FUNCTION_BLOCK FB_MqttLight EXTENDS FB_Light IMPLEMENTS I_MqttMessageReceiver, I_MqttDeviceDiscoveryProvider
VAR_INPUT
END_VAR
VAR_OUTPUT
END_VAR
VAR
	rMqttController: REFERENCE TO FB_MqttController;
	fbDeviceDiscovery : FB_MqttLightDiscovery;
	sStateTopic: STRING(255); // The topic to publish the state to
	sCommandTopic : STRING(255);
	sCmdOnPayload: STRING(10); // The text which is published if On() is called
	sCmdOffPayload: STRING(10); // The test which is published if Off() is called
	sStateOnPayload: STRING(10); // The text which is published if On() is called
	sStateOffPayload: STRING(10); // The test which is published if Off() is called
END_VAR

METHOD FB_init : BOOL
VAR_INPUT
	bInitRetains : BOOL; // if TRUE, the retain variables are initialized (warm start / cold start)
	bInCopyCode : BOOL;  // if TRUE, the instance afterwards gets moved into the copy code (online change)
	rMqttController : REFERENCE TO FB_MqttController;
	sMainTopic : STRING(255); // The topic to publish
	sIdentifier : STRING(20);
	sName : STRING(30);
END_VAR
VAR
	stDevInfo : ST_MqttDeviceInformation;
	stDevConfig : ST_MqttLightConfiguration;
END_VAR
THIS^.rMqttController REF= rMqttController;

THIS^.sStateTopic := CONCAT(STR1 := sMainTopic, STR2 := '/');
THIS^.sStateTopic := CONCAT(STR1 := THIS^.sStateTopic, STR2 := GVL_MQTT_CONST.TOPIC_STATE);
THIS^.sCommandTopic := CONCAT(STR1 := sMainTopic, STR2 := '/');
THIS^.sCommandTopic := CONCAT(STR1 := THIS^.sCommandTopic, STR2 := GVL_MQTT_CONST.TOPIC_COMMAND);

THIS^.fbDeviceDiscovery.SetMqttClient(rMqttClient := THIS^.rMqttController.MqttClient);
THIS^.fbDeviceDiscovery.NodeId := GVL_MQTT_CONST.DEV_DISCOVER_NODEID;
THIS^.fbDeviceDiscovery.ObjectId := sIdentifier;

stDevConfig.command_topic := THIS^.sCommandTopic;
stDevConfig.state_topic := THIS^.sStateTopic;
stDevConfig.unique_id := sIdentifier;
stDevConfig.name := sName;
THIS^.fbDeviceDiscovery.Configuration := stDevConfig;

stDevInfo.identifiers := sIdentifier;
stDevInfo.manufacturer := GVL_MQTT_CONST.DEV_DISCOVER_MANUFACTURER;
stDevInfo.model := 'FB_MqttLight';
stDevInfo.sw_version := GVL_CONST.SW_VERSION;
stDevInfo.name := sName;
THIS^.fbDeviceDiscovery.DeviceInformation := stDevInfo;

THIS^.rMqttController.RegisterMqttMessageReceive(iMqttMessageReceiver := THIS^, sTopic := sCommandTopic);
THIS^.sCmdOnPayload := GVL_MQTT_CONST.PL_LIGHT_COMMAND_ON;
THIS^.sCmdOffPayload := GVL_MQTT_CONST.PL_LIGHT_COMMAND_OFF;
THIS^.sStateOnPayload := GVL_MQTT_CONST.PL_LIGHT_STATE_ON;
THIS^.sStateOffPayload := GVL_MQTT_CONST.PL_LIGHT_STATE_OFF;
END_METHOD

METHOD GetMqttDeviceDiscovery : I_MqttDeviceDiscovery
VAR_INPUT
END_VAR
GetMqttDeviceDiscovery := this^.fbDeviceDiscovery;
END_METHOD

METHOD Off : BOOL
SUPER^.Off();
THIS^.SendStatus();
END_METHOD

METHOD On : BOOL
SUPER^.On();
THIS^.SendStatus();
END_METHOD

METHOD OnMqttMessage : BOOL
VAR_INPUT
	rMqttMessage : REFERENCE TO FB_IotMqttMessage;
END_VAR
VAR
	sPayload : STRING(10);
	bSuccess : BOOL := FALSE;
END_VAR
IF (__ISVALIDREF(rMqttMessage)) THEN
	IF rMqttMessage.GetPayload(pPayload := ADR(sPayload),
			nPayloadSize := 10,
			bSetNullTermination := TRUE) THEN
		IF F_StrCmp(pStr1 := ADR(sPayload), pStr2 := ADR(THIS^.sCmdOnPayload)) THEN
			THIS^.On();
			bSuccess := TRUE;
		ELSIF F_StrCmp(pStr1 := ADR(sPayload), pStr2 := ADR(THIS^.sCmdOffPayload)) THEN
			THIS^.Off();
			bSuccess := TRUE;
		END_IF
	END_IF
END_IF

OnMqttMessage := bSuccess;
END_METHOD

METHOD PRIVATE SendStatus : BOOL
VAR_INPUT
END_VAR
VAR
	sStatus : STRING(10);
END_VAR
IF (__ISVALIDREF(rMqttController) AND __ISVALIDREF(rMqttController.MqttClient)) THEN
	IF (rMqttController.MqttClient.bConnected) THEN
		IF Active THEN
			sStatus := sStateOnPayload;
		ELSE
			sStatus := sStateOffPayload;
		END_IF
		rMqttController.MqttClient.Publish(sTopic:= sStateTopic, 
			pPayload:= ADR(sStatus), nPayloadSize:= LEN2(ADR(sStatus)),
			eQoS:= TcIotMqttQos.AtLeastOnceDelivery, bRetain:= TRUE,
			bQueue:= FALSE);
	END_IF
END_IF
END_METHOD

END_FUNCTION_BLOCK

(* stored: Version 1.1.0.1, ProductVersion 3.1.4024.5
   POU FB_MqttLight: Id {6ebf0452-2f75-444e-81f6-69cd58362e1d}, SpecialFunc None
   Method FB_init: Id {d0dff497-1b25-4b88-be14-73174c0961cf}
   Method GetMqttDeviceDiscovery: Id {3be87e2a-d266-408f-b2cb-b557a06b1419}
   Method Off: Id {6468975b-7258-4f68-a05c-0a86da40a0e4}
   Method On: Id {b6ca792a-382b-486d-974e-7e4a9442e530}
   Method OnMqttMessage: Id {ad538b84-229a-42d7-81c4-02f2e5e5fe70}
   Method SendStatus: Id {24f70da2-24c1-4861-a1e8-abd502fc6cfc} *)
